// TwinCAT 3 PLC project PLC
// ProgramVersion: 3.1.4026.26
// libraries:
//   Tc2_Standard, * (Beckhoff Automation GmbH)
//   Tc2_System, * (Beckhoff Automation GmbH)
// project tree:
//   / PlcTask.TcTTO
//   POUs/ MAIN.TcPOU
// real-time tasks:
//   TASK PlcTask: cycle T#10ms, priority 20, ADS port 350
//   TASK PNTask: cycle T#1ms, priority 1, ADS port 301
//   TASK PNTaskDevice: cycle T#2ms, priority 2, ADS port 302
// I/O:
//   DEVICE Device 1 (EtherCAT), AmsNetId 5.162.174.122.2.1
//     Term 1 (EK1200) [EK1200-5000 EtherCAT Power supply (2A E-Bus)]
//       Term 2 (EL6631-0010) [EL6631-0010 PROFINET IO Device]
//       Term 3 (EL9011)
//   DEVICE Device 3 (Profinet Controller CCAT (RT)), AmsNetId 5.162.174.122.4.1
//     el6631-0010 [Beckhoff Automation PROFINET I/O device - EtherCAT slave terminal, V2.0 EL6631-0010]
//       modules: Term 1 (DAP Module), Term 2 (1 Word In- and Output), Term 3 (1 Word In- and Output)
// variable links:
//   (this object) <-> Device 1 (EtherCAT)
//     PlcTask Inputs/MAIN.DevState <-> Inputs/DevState
//   (this object) <-> Device 3 (Profinet Controller CCAT (RT))/el6631-0010
//     PlcTask Inputs/MAIN.b_CtrlIn[0] <-> API/Term 2 (1 Word In- and Output)/Subterm 2 (1 Word In- and Output)/Inputs/1 Word Input
//     PlcTask Inputs/MAIN.b_CtrlIn[1] <-> API/Term 3 (1 Word In- and Output)/Subterm 3 (1 Word In- and Output)/Inputs/1 Word Input
//     PlcTask Outputs/MAIN.b_CtrlOut[0] <-> API/Term 2 (1 Word In- and Output)/Subterm 2 (1 Word In- and Output)/Outputs/1 Word Output
//     PlcTask Outputs/MAIN.b_CtrlOut[1] <-> API/Term 3 (1 Word In- and Output)/Subterm 3 (1 Word In- and Output)/Outputs/1 Word Output

CONFIGURATION PLC
    RESOURCE PLC ON TwinCAT3
        TASK PlcTask(INTERVAL := T#10ms, PRIORITY := 20);
        PROGRAM MAIN WITH PlcTask : MAIN;
    END_RESOURCE
END_CONFIGURATION

// ---- POUs/MAIN.TcPOU
PROGRAM MAIN
VAR
	DevState  AT %I* : UINT;
	{attribute 'OPC.UA.DA' := '1'}
	ContadorOpcUa : DINT := 0;
    // Variáveis do lado Controller (Envia dados)
    b_CtrlOut  AT %Q* : ARRAY[0..1] OF WORD;
    b_CtrlIn   AT %I* : ARRAY[0..1] OF WORD;

    // Variáveis do lado Device (Recebe e processa)
    b_DevIn    AT %I* : ARRAY[0..1] OF WORD;
    b_DevOut   AT %Q* : ARRAY[0..1] OF WORD;

    // Contador para o teste
    u_Counter         : WORD := 0;
END_VAR

// 1. Controller incrementa um contador e envia para a rede
u_Counter := u_Counter + 1;
b_CtrlOut[0] := u_Counter;

// 2. Lógica de Eco/Loopback no Device (Pega o que entrou e joga na saída)
b_DevOut[0] := b_DevIn[0];

ContadorOpcUa := ContadorOpcUa + 1;

END_PROGRAM
